{attribute 'qualified_only'}
VAR_GLOBAL
    // Pitch Mechanism:
    {attribute 'TcLinkTo' := '.diEncCnt:=TIIB[EL5042_M1L0_PitchBender]^FB Inputs Channel 1^Position'}
    M1L0_Pitch : HOMS_PitchMechanism := (ReqPosLimHi := 120.0,
                                         ReqPosLimLo := -182.0,
                                         diEncPosLimHi := 8662020,
                                         diEncPosLimLo := 8507095);
    // M1L0 Flow Press Sensors
    {attribute 'TcLinkTo' := '.iRaw := TIIB[EL3054_M1L0_FWM_PRSM]^AI Standard Channel 1^Value'}
    fM1L0_Flow_1 : FB_AnalogInput;
    {attribute 'pytmc' := '
        pv: MR1L0:HOMS:FWM:1
        field: EGU lpm
        io: i
    '}
    fM1L0_Flow_1_val : LREAL;
    {attribute 'TcLinkTo' := '.iRaw := TIIB[EL3054_M1L0_FWM_PRSM]^AI Standard Channel 2^Value'}
    fM1L0_Flow_2 : FB_AnalogInput;
    {attribute 'pytmc' := '
        pv: MR1L0:HOMS:FWM:2
        field: EGU lpm
        io: i
    '}
    fM1L0_Flow_2_val : LREAL;
    {attribute 'TcLinkTo' := '.iRaw := TIIB[EL3054_M1L0_FWM_PRSM]^AI Standard Channel 3^Value'}
    fM1L0_Press_1 : FB_AnalogInput;
    {attribute 'pytmc' := '
        pv: MR1L0:HOMS:PRSM:1
        field: EGU bar
        io: i
    '}
    fM1L0_Press_1_val : LREAL;
END_VAR

(* stored: Version 1.1.0.1, ProductVersion 3.1.4022.18
   GVL GVL_M1L0: Id {c3e91af1-5ac0-497f-aea6-a43e8c284355} *)
